Staubli VAL3: StepMove.pgx

public program StepMove(num x_nAxisNum, num x_nKey, bool x_bJog)
begin
  //
  if isKeyPressed(x_nKey)
    //x_bjog=true:正向运动
    if x_bJog
      ? "+"
      aioSet(aoWorkMode[x_nAxisNum],-1)
      doStartHoming[x_nAxisNum]=true
    else
      ? "-"
      aioSet(aoWorkMode[x_nAxisNum],-1)
      doManual[x_nAxisNum]=true
    endIf
    wait(isKeyPressed(x_nKey)==false)
  else
    doStartHoming[x_nAxisNum]=false
    doManual[x_nAxisNum]=false
  endIf
end
